# EPICS autosave request: ip/ipApp/Db/SR830_settings.req
# FILE... SR830_settings.req
$(P)SR830:$(N):read.DESC
$(P)SR830:$(N):TC1
$(P)SR830:$(N):TC2
$(P)SR830:$(N):TC3
$(P)SR830:$(N):FiltCh
$(P)SR830:$(N):Sens1
$(P)SR830:$(N):Sens2
$(P)SR830:$(N):Sens3
$(P)SR830:$(N):ResvCh
$(P)SR830:$(N):Disp1Ch
$(P)SR830:$(N):Disp2Ch
$(P)SR830:$(N):Disp3Ch
$(P)SR830:$(N):read.SCAN
$(P)SR830:$(N):SetPhas.A
$(P)SR830:$(N):SetFreq.A
$(P)SR830:$(N):SetAmpl.A
